FUNCTION_BLOCK PAMDryer EXTENDS PAProcessModule
VAR_INPUT
END_VAR
VAR_OUTPUT
END_VAR
VAR
	_PAPointMatIn1 : PAPoint(THIS^);
	_PAPointMatOut1 : PAPoint(THIS^);
END_VAR

METHOD FB_init : BOOL
VAR_INPUT
	bInitRetains : BOOL; // if TRUE, the retain variables are initialized (warm start / cold start)
	bInCopyCode : BOOL;  // if TRUE, the instance afterwards gets moved into the copy code (online change)
	parent : IACComponent;
END_VAR
AddPoint(_PAPointMatIn1);
AddPoint(_PAPointMatOut1);
END_METHOD

PROPERTY PUBLIC PAPointMatIn1 : IACPoint
GET
PAPointMatIn1 := _PAPointMatIn1;
END_GET
END_PROPERTY

PROPERTY PUBLIC PAPointMatOut1 : IACPoint
GET
PAPointMatOut1 := _PAPointMatOut1;
END_GET
END_PROPERTY

END_FUNCTION_BLOCK

(* stored: Version 1.1.0.1, ProductVersion 3.1.4020.12
   POU PAMDryer: Id {0d1f780d-962a-431e-a16a-2162aa62aa7a}, SpecialFunc None
   Method FB_init: Id {ad93020e-648e-4f10-b3e2-cc7c758b48c8}
   Property PAPointMatIn1: Id {58f00a77-d489-4421-ad65-0f053d00a5c7}
   Get Get: Id {61140c23-049a-4a45-9288-0a50befb9461}
   Property PAPointMatOut1: Id {89506cae-3753-410c-a77a-89839a9f647f}
   Get Get: Id {86a42e61-3acf-449e-b918-d95db4682991} *)
